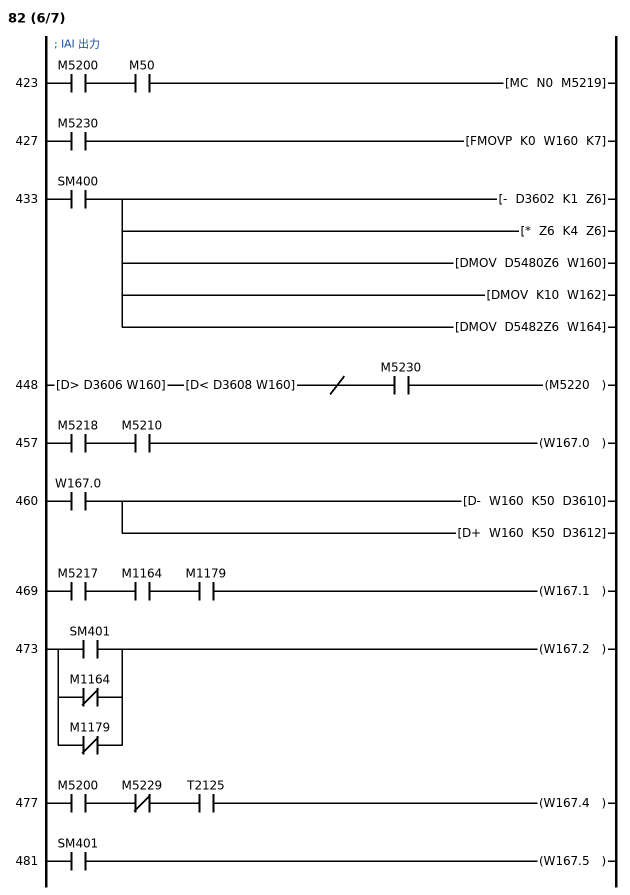
; IAI 出力
423   LD      M5200
      AND     M50
      MC      N0 M5219
427   LD      M5230
      FMOVP   K0 W160 K7
433   LD      SM400
      -       D3602 K1 Z6
      *       Z6 K4 Z6
      DMOV    D5480Z6 W160
      DMOV    K10 W162
      DMOV    D5482Z6 W164
448   LDD>    D3606 W160
      ANDD<   D3608 W160
      INV
      AND     M5230
      OUT     M5220
457   LD      M5218
      AND     M5210
      OUT     W167.0
460   LD      W167.0
      D-      W160 K50 D3610
      D+      W160 K50 D3612
469   LD      M5217
      AND     M1164
      AND     M1179
      OUT     W167.1
473   LD      SM401
      ORI     M1164
      ORI     M1179
      OUT     W167.2
477   LD      M5200
      ANI     M5229
      AND     T2125
      OUT     W167.4
481   LD      SM401
      OUT     W167.5
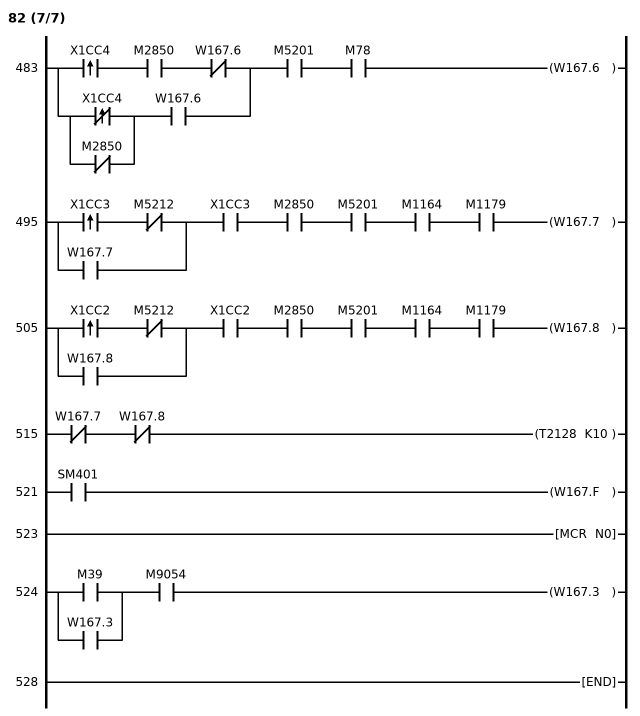
483   LDP     X1CC4
      AND     M2850
      ANI     W167.6
      LDPI    X1CC4
      ORI     M2850
      AND     W167.6
      ORB
      AND     M5201
      AND     M78
      OUT     W167.6
495   LDP     X1CC3
      ANI     M5212
      OR      W167.7
      AND     X1CC3
      AND     M2850
      AND     M5201
      AND     M1164
      AND     M1179
      OUT     W167.7
505   LDP     X1CC2
      ANI     M5212
      OR      W167.8
      AND     X1CC2
      AND     M2850
      AND     M5201
      AND     M1164
      AND     M1179
      OUT     W167.8
515   LDI     W167.7
      ANI     W167.8
      OUT     T2128 K10
521   LD      SM401
      OUT     W167.F
523   MCR     N0
524   LD      M39
      OR      W167.3
      AND     M9054
      OUT     W167.3
528   END
END_PROGRAM

PROGRAM 83
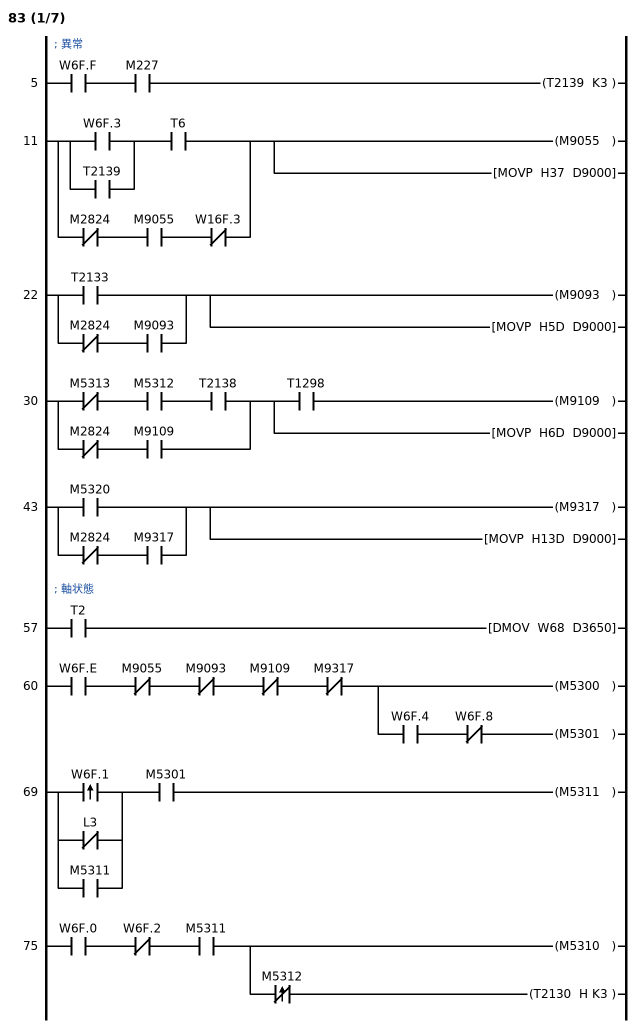
; 異常
5     LD      W6F.F
      AND     M227
      OUT     T2139 K3
11    LD      W6F.3
      OR      T2139
      AND     T6
      LDI     M2824
      AND     M9055
      ANI     W16F.3
      ORB
      OUT     M9055
      MOVP    H37 D9000
22    LD      T2133
      LDI     M2824
      AND     M9093
      ORB
      OUT     M9093
      MOVP    H5D D9000
30    LDI     M5313
      AND     M5312
      AND     T2138
      LDI     M2824
      AND     M9109
      ORB
      MPS
      AND     T1298
      OUT     M9109
      MPP
      MOVP    H6D D9000
43    LD      M5320
      LDI     M2824
      AND     M9317
      ORB
      OUT     M9317
      MOVP    H13D D9000
; 軸状態
57    LD      T2
      DMOV    W68 D3650
60    LD      W6F.E
      ANI     M9055
      ANI     M9093
      ANI     M9109
      ANI     M9317
      OUT     M5300
      AND     W6F.4
      ANI     W6F.8
      OUT     M5301
69    LDP     W6F.1
      ORI     L3
      OR      M5311
      AND     M5301
      OUT     M5311
75    LD      W6F.0
      ANI     W6F.2
      AND     M5311
      OUT     M5310
      ANDPI   M5312
      OUTH    T2130 K3
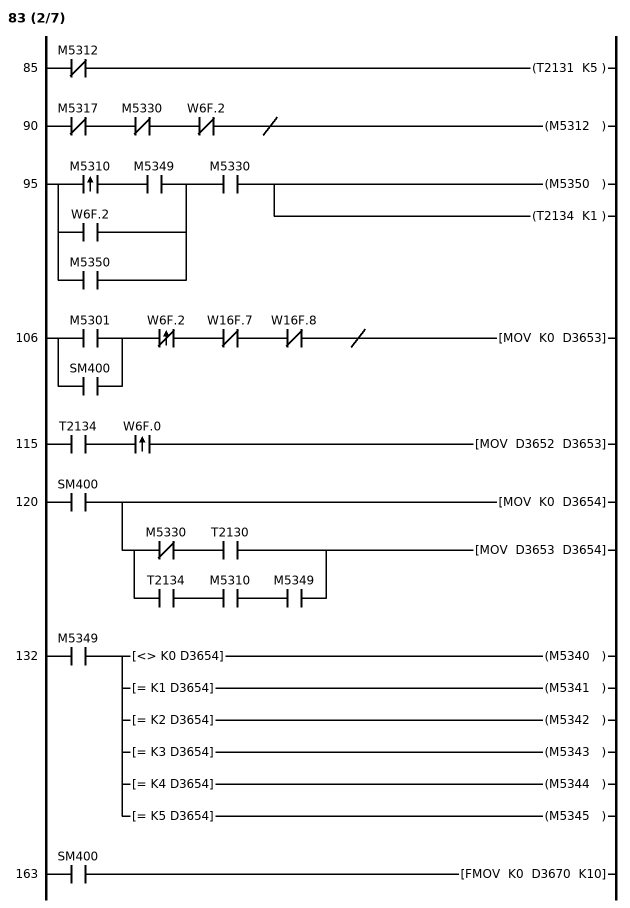
85    LDI     M5312
      OUT     T2131 K5
90    LDI     M5317
      ANI     M5330
      ANI     W6F.2
      INV
      OUT     M5312
95    LDP     M5310
      AND     M5349
      OR      W6F.2
      OR      M5350
      AND     M5330
      OUT     M5350
      OUT     T2134 K1
106   LD      M5301
      OR      SM400
      ANDPI   W6F.2
      ANI     W16F.7
      ANI     W16F.8
      INV
      MOV     K0 D3653
115   LD      T2134
      ANDP    W6F.0
      MOV     D3652 D3653
120   LD      SM400
      MOV     K0 D3654
      LDI     M5330
      AND     T2130
      LD      T2134
      AND     M5310
      AND     M5349
      ORB
      ANB
      MOV     D3653 D3654
132   LD      M5349
      MPS
      AND<>   K0 D3654
      OUT     M5340
      MRD
      AND=    K1 D3654
      OUT     M5341
      MRD
      AND=    K2 D3654
      OUT     M5342
      MRD
      AND=    K3 D3654
      OUT     M5343
      MRD
      AND=    K4 D3654
      OUT     M5344
      MPP
      AND=    K5 D3654
      OUT     M5345
163   LD      SM400
      FMOV    K0 D3670 K10
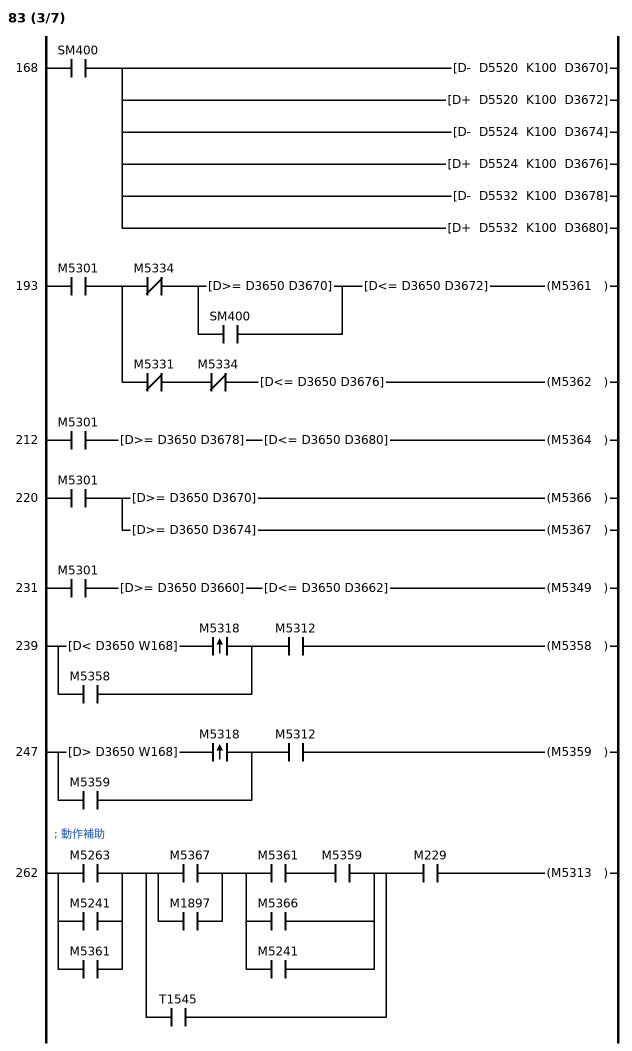
168   LD      SM400
      D-      D5520 K100 D3670
      D+      D5520 K100 D3672
      D-      D5524 K100 D3674
      D+      D5524 K100 D3676
      D-      D5532 K100 D3678
      D+      D5532 K100 D3680
193   LD      M5301
      MPS
      ANI     M5334
      LDD>=   D3650 D3670
      OR      SM400
      ANB
      ANDD<=  D3650 D3672
      OUT     M5361
      MPP
      ANI     M5331
      ANI     M5334
      ANDD<=  D3650 D3676
      OUT     M5362
212   LD      M5301
      ANDD>=  D3650 D3678
      ANDD<=  D3650 D3680
      OUT     M5364
220   LD      M5301
      MPS
      ANDD>=  D3650 D3670
      OUT     M5366
      MPP
      ANDD>=  D3650 D3674
      OUT     M5367
231   LD      M5301
      ANDD>=  D3650 D3660
      ANDD<=  D3650 D3662
      OUT     M5349
239   LDD<    D3650 W168
      ANDP    M5318
      OR      M5358
      AND     M5312
      OUT     M5358
247   LDD>    D3650 W168
      ANDP    M5318
      OR      M5359
      AND     M5312
      OUT     M5359
; 動作補助
262   LD      M5263
      OR      M5241
      OR      M5361
      LD      M5367
      OR      M1897
      LD      M5361
      AND     M5359
      OR      M5366
      OR      M5241
      ANB
      OR      T1545
      ANB
      AND     M229
      OUT     M5313
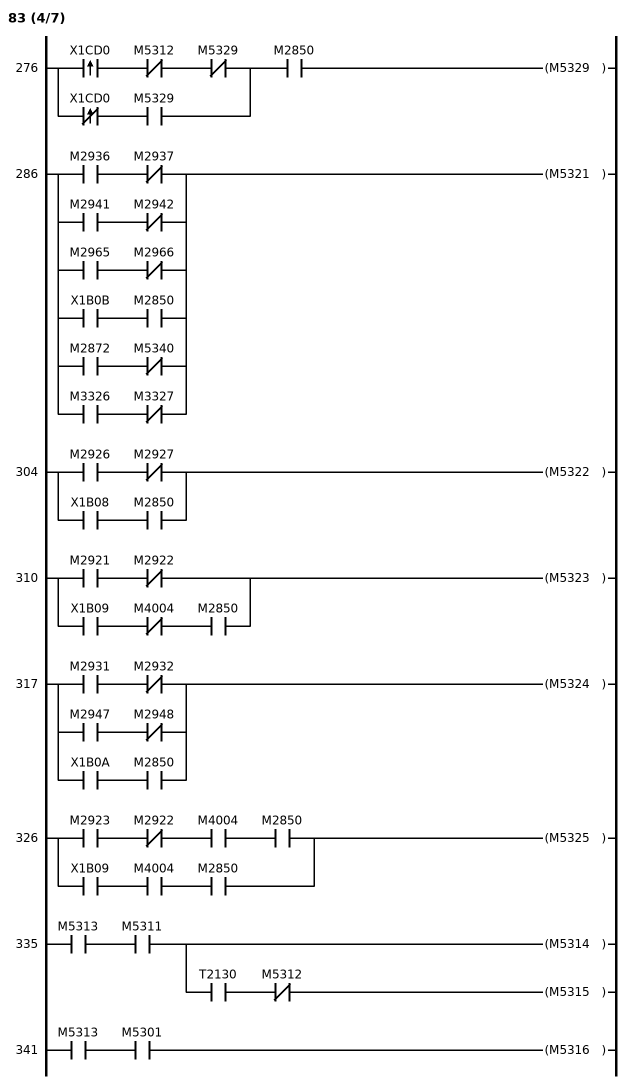
276   LDP     X1CD0
      ANI     M5312
      ANI     M5329
      LDPI    X1CD0
      AND     M5329
      ORB
      AND     M2850
      OUT     M5329
286   LD      M2936
      ANI     M2937
      LD      M2941
      ANI     M2942
      ORB
      LD      M2965
      ANI     M2966
      ORB
      LD      X1B0B
      AND     M2850
      ORB
      LD      M2872
      ANI     M5340
      ORB
      LD      M3326
      ANI     M3327
      ORB
      OUT     M5321
304   LD      M2926
      ANI     M2927
      LD      X1B08
      AND     M2850
      ORB
      OUT     M5322
310   LD      M2921
      ANI     M2922
      LD      X1B09
      ANI     M4004
      AND     M2850
      ORB
      OUT     M5323
317   LD      M2931
      ANI     M2932
      LD      M2947
      ANI     M2948
      ORB
      LD      X1B0A
      AND     M2850
      ORB
      OUT     M5324
326   LD      M2923
      ANI     M2922
      AND     M4004
      AND     M2850
      LD      X1B09
      AND     M4004
      AND     M2850
      ORB
      OUT     M5325
335   LD      M5313
      AND     M5311
      OUT     M5314
      AND     T2130
      ANI     M5312
      OUT     M5315
341   LD      M5313
      AND     M5301
      OUT     M5316
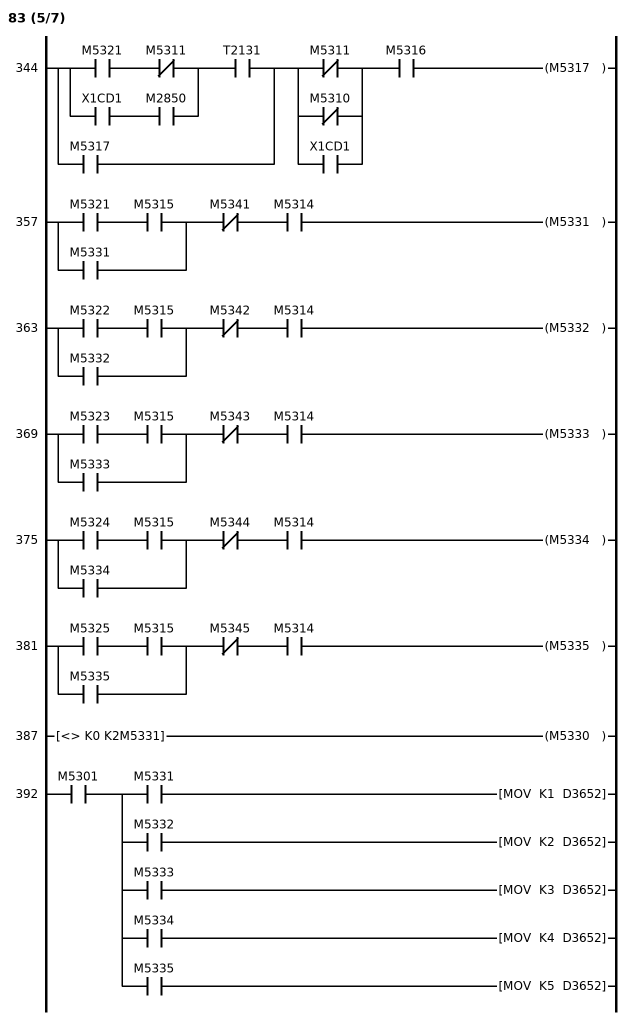
344   LD      M5321
      ANI     M5311
      LD      X1CD1
      AND     M2850
      ORB
      AND     T2131
      OR      M5317
      LDI     M5311
      ORI     M5310
      OR      X1CD1
      ANB
      AND     M5316
      OUT     M5317
357   LD      M5321
      AND     M5315
      OR      M5331
      ANI     M5341
      AND     M5314
      OUT     M5331
363   LD      M5322
      AND     M5315
      OR      M5332
      ANI     M5342
      AND     M5314
      OUT     M5332
369   LD      M5323
      AND     M5315
      OR      M5333
      ANI     M5343
      AND     M5314
      OUT     M5333
375   LD      M5324
      AND     M5315
      OR      M5334
      ANI     M5344
      AND     M5314
      OUT     M5334
381   LD      M5325
      AND     M5315
      OR      M5335
      ANI     M5345
      AND     M5314
      OUT     M5335
387   LD<>    K0 K2M5331
      OUT     M5330
392   LD      M5301
      MPS
      AND     M5331
      MOV     K1 D3652
      MRD
      AND     M5332
      MOV     K2 D3652
      MRD
      AND     M5333
      MOV     K3 D3652
      MRD
      AND     M5334
      MOV     K4 D3652
      MPP
      AND     M5335
      MOV     K5 D3652
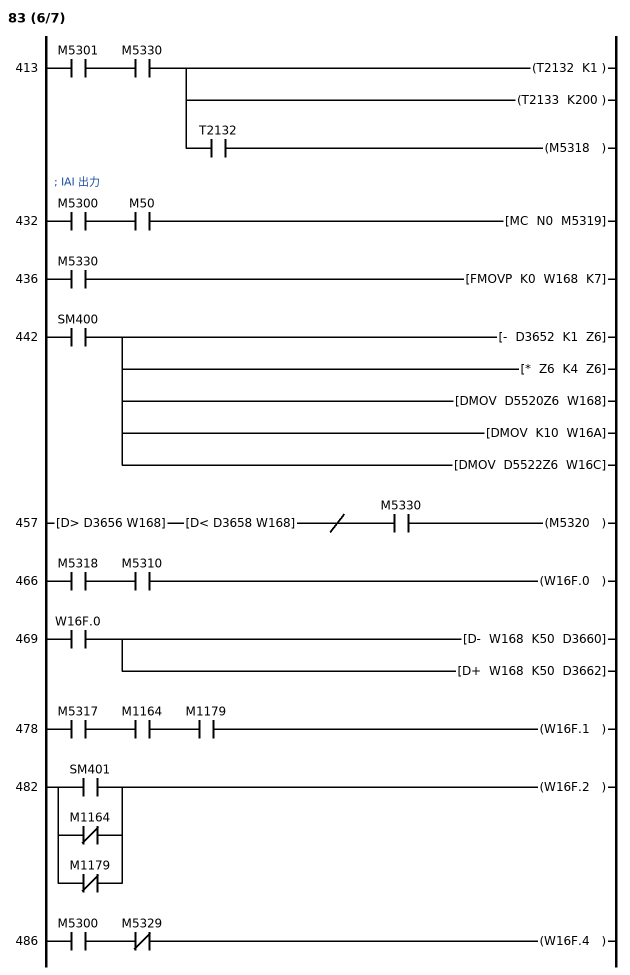
413   LD      M5301
      AND     M5330
      OUT     T2132 K1
      OUT     T2133 K200
      AND     T2132
      OUT     M5318
; IAI 出力
432   LD      M5300
      AND     M50
      MC      N0 M5319
436   LD      M5330
      FMOVP   K0 W168 K7
442   LD      SM400
      -       D3652 K1 Z6
      *       Z6 K4 Z6
      DMOV    D5520Z6 W168
      DMOV    K10 W16A
      DMOV    D5522Z6 W16C
457   LDD>    D3656 W168
      ANDD<   D3658 W168
      INV
      AND     M5330
      OUT     M5320
466   LD      M5318
      AND     M5310
      OUT     W16F.0
469   LD      W16F.0
      D-      W168 K50 D3660
      D+      W168 K50 D3662
478   LD      M5317
      AND     M1164
      AND     M1179
      OUT     W16F.1
482   LD      SM401
      ORI     M1164
      ORI     M1179
      OUT     W16F.2
486   LD      M5300
      ANI     M5329
      OUT     W16F.4
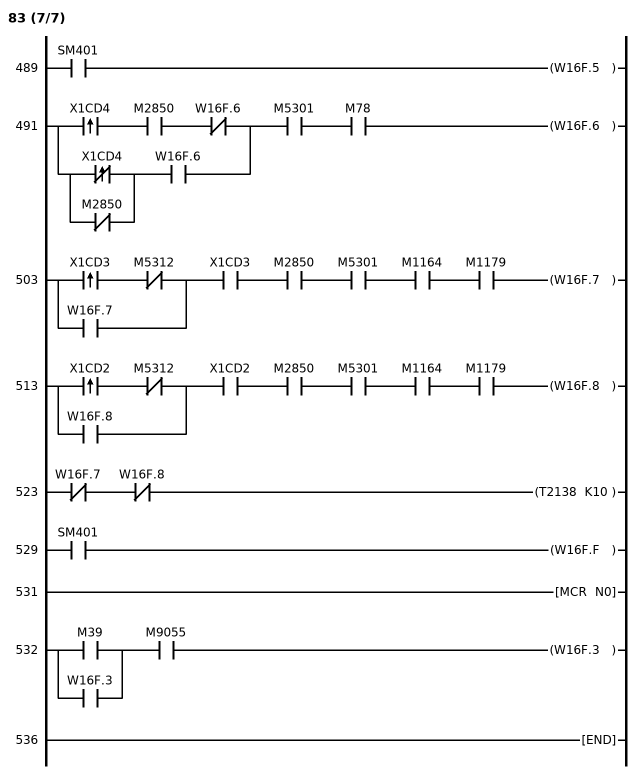
489   LD      SM401
      OUT     W16F.5
491   LDP     X1CD4
      AND     M2850
      ANI     W16F.6
      LDPI    X1CD4
      ORI     M2850
      AND     W16F.6
      ORB
      AND     M5301
      AND     M78
      OUT     W16F.6
503   LDP     X1CD3
      ANI     M5312
      OR      W16F.7
      AND     X1CD3
      AND     M2850
      AND     M5301
      AND     M1164
      AND     M1179
      OUT     W16F.7
513   LDP     X1CD2
      ANI     M5312
      OR      W16F.8
      AND     X1CD2
      AND     M2850
      AND     M5301
      AND     M1164
      AND     M1179
      OUT     W16F.8
523   LDI     W16F.7
      ANI     W16F.8
      OUT     T2138 K10
529   LD      SM401
      OUT     W16F.F
531   MCR     N0
532   LD      M39
      OR      W16F.3
      AND     M9055
      OUT     W16F.3
536   END
END_PROGRAM

PROGRAM 90
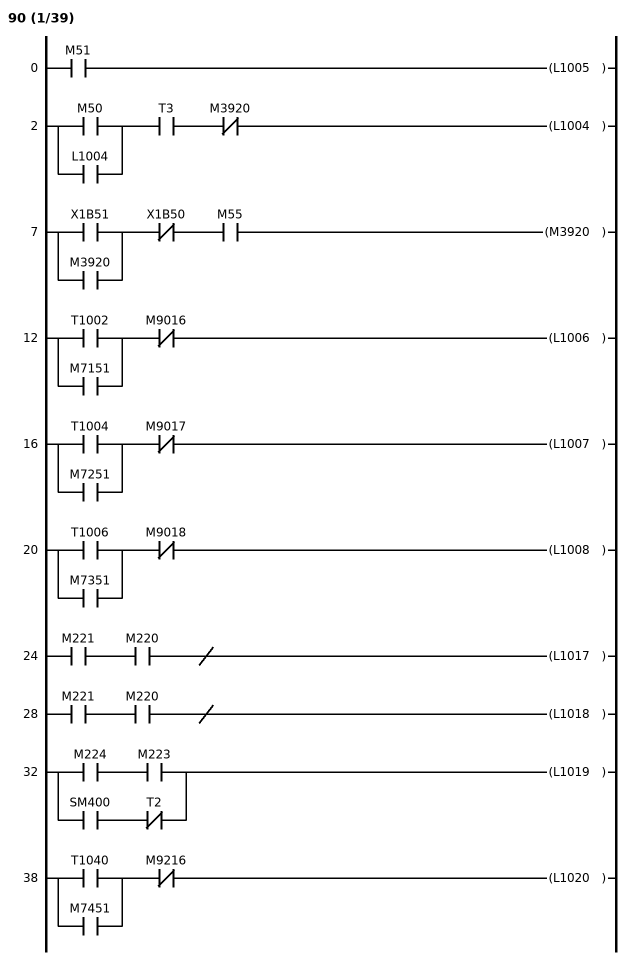
0     LD      M51
      OUT     L1005
2     LD      M50
      OR      L1004
      AND     T3
      ANI     M3920
      OUT     L1004
7     LD      X1B51
      OR      M3920
      ANI     X1B50
      AND     M55
      OUT     M3920
12    LD      T1002
      OR      M7151
      ANI     M9016
      OUT     L1006
16    LD      T1004
      OR      M7251
      ANI     M9017
      OUT     L1007
20    LD      T1006
      OR      M7351
      ANI     M9018
      OUT     L1008
24    LD      M221
      AND     M220
      INV
      OUT     L1017
28    LD      M221
      AND     M220
      INV
      OUT     L1018
32    LD      M224
      AND     M223
      LD      SM400
      ANI     T2
      ORB
      OUT     L1019
38    LD      T1040
      OR      M7451
      ANI     M9216
      OUT     L1020
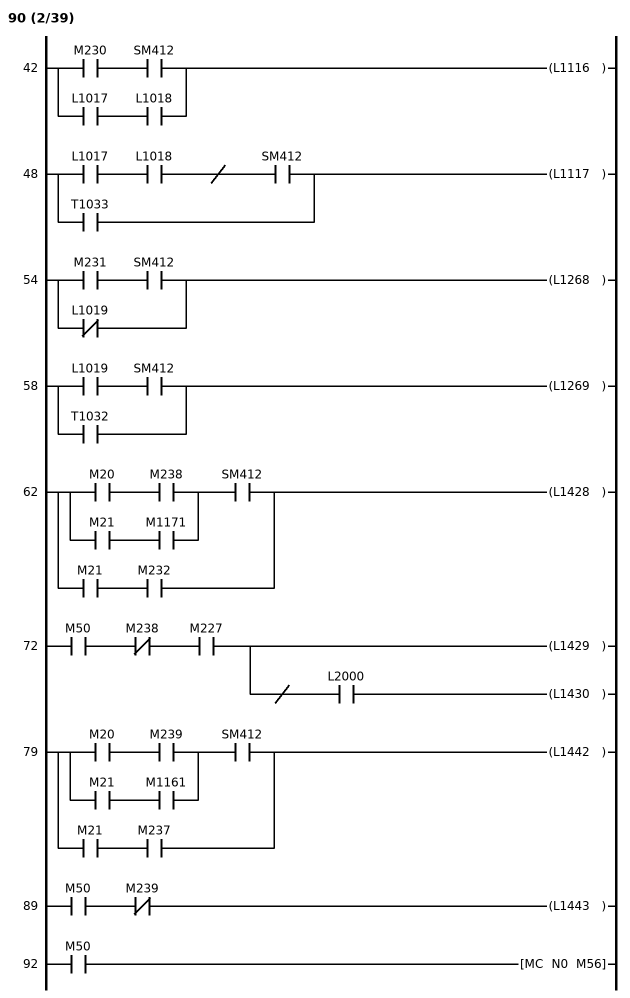
42    LD      M230
      AND     SM412
      LD      L1017
      AND     L1018
      ORB
      OUT     L1116
48    LD      L1017
      AND     L1018
      INV
      AND     SM412
      OR      T1033
      OUT     L1117
54    LD      M231
      AND     SM412
      ORI     L1019
      OUT     L1268
58    LD      L1019
      AND     SM412
      OR      T1032
      OUT     L1269
62    LD      M20
      AND     M238
      LD      M21
      AND     M1171
      ORB
      AND     SM412
      LD      M21
      AND     M232
      ORB
      OUT     L1428
72    LD      M50
      ANI     M238
      AND     M227
      OUT     L1429
      INV
      AND     L2000
      OUT     L1430
79    LD      M20
      AND     M239
      LD      M21
      AND     M1161
      ORB
      AND     SM412
      LD      M21
      AND     M237
      ORB
      OUT     L1442
89    LD      M50
      ANI     M239
      OUT     L1443
92    LD      M50
      MC      N0 M56
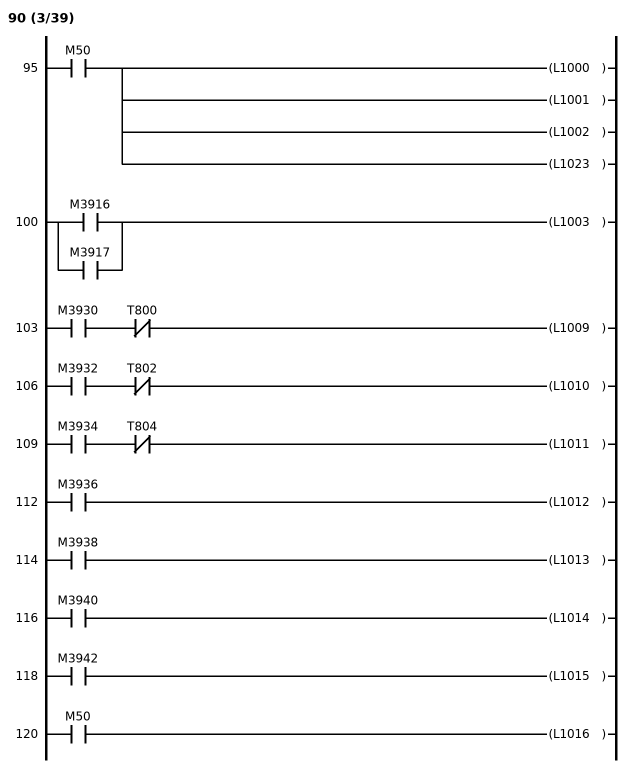
95    LD      M50
      OUT     L1000
      OUT     L1001
      OUT     L1002
      OUT     L1023
100   LD      M3916
      OR      M3917
      OUT     L1003
103   LD      M3930
      ANI     T800
      OUT     L1009
106   LD      M3932
      ANI     T802
      OUT     L1010
109   LD      M3934
      ANI     T804
      OUT     L1011
112   LD      M3936
      OUT     L1012
114   LD      M3938
      OUT     L1013
116   LD      M3940
      OUT     L1014
118   LD      M3942
      OUT     L1015
120   LD      M50
      OUT     L1016
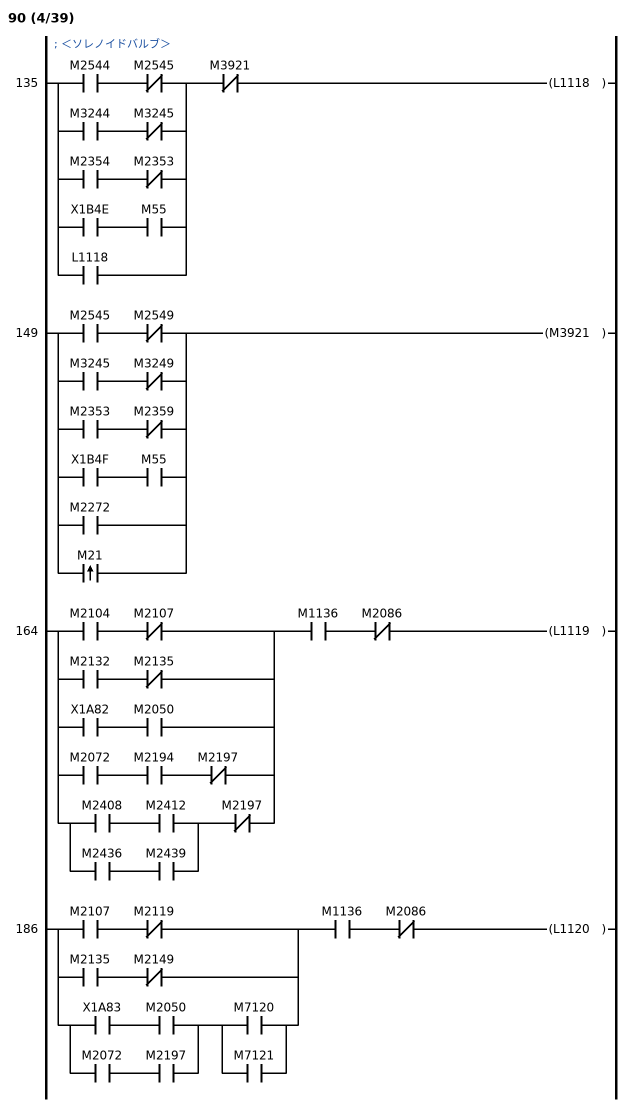
; ＜ソレノイドバルブ＞
135   LD      M2544
      ANI     M2545
      LD      M3244
      ANI     M3245
      ORB
      LD      M2354
      ANI     M2353
      ORB
      LD      X1B4E
      AND     M55
      ORB
      OR      L1118
      ANI     M3921
      OUT     L1118
149   LD      M2545
      ANI     M2549
      LD      M3245
      ANI     M3249
      ORB
      LD      M2353
      ANI     M2359
      ORB
      LD      X1B4F
      AND     M55
      ORB
      OR      M2272
      ORP     M21
      OUT     M3921
164   LD      M2104
      ANI     M2107
      LD      M2132
      ANI     M2135
      ORB
      LD      X1A82
      AND     M2050
      ORB
      LD      M2072
      AND     M2194
      ANI     M2197
      ORB
      LD      M2408
      AND     M2412
      LD      M2436
      AND     M2439
      ORB
      ANI     M2197
      ORB
      AND     M1136
      ANI     M2086
      OUT     L1119
186   LD      M2107
      ANI     M2119
      LD      M2135
      ANI     M2149
      ORB
      LD      X1A83
      AND     M2050
      LD      M2072
      AND     M2197
      ORB
      LD      M7120
      OR      M7121
      ANB
      ORB
      AND     M1136
      ANI     M2086
      OUT     L1120
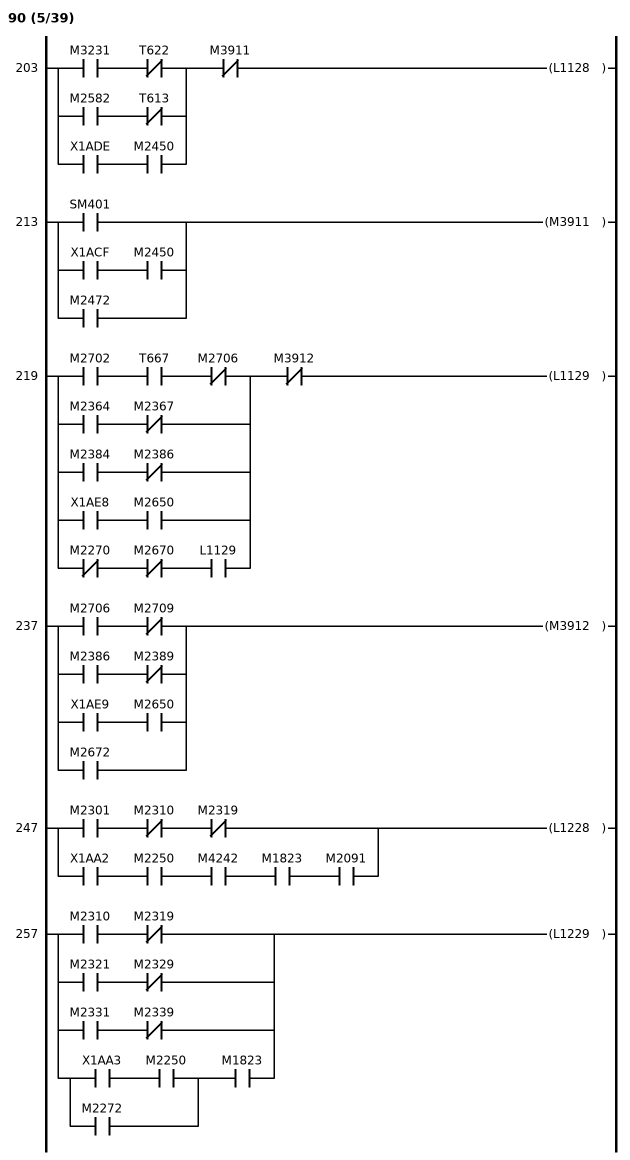
203   LD      M3231
      ANI     T622
      LD      M2582
      ANI     T613
      ORB
      LD      X1ADE
      AND     M2450
      ORB
      ANI     M3911
      OUT     L1128
213   LD      SM401
      LD      X1ACF
      AND     M2450
      ORB
      OR      M2472
      OUT     M3911
219   LD      M2702
      AND     T667
      ANI     M2706
      LD      M2364
      ANI     M2367
      ORB
      LD      M2384
      ANI     M2386
      ORB
      LD      X1AE8
      AND     M2650
      ORB
      LDI     M2270
      ANI     M2670
      AND     L1129
      ORB
      ANI     M3912
      OUT     L1129
237   LD      M2706
      ANI     M2709
      LD      M2386
      ANI     M2389
      ORB
      LD      X1AE9
      AND     M2650
      ORB
      OR      M2672
      OUT     M3912
247   LD      M2301
      ANI     M2310
      ANI     M2319
      LD      X1AA2
      AND     M2250
      AND     M4242
      AND     M1823
      AND     M2091
      ORB
      OUT     L1228
257   LD      M2310
      ANI     M2319
      LD      M2321
      ANI     M2329
      ORB
      LD      M2331
      ANI     M2339
      ORB
      LD      X1AA3
      AND     M2250
      OR      M2272
      AND     M1823
      ORB
      OUT     L1229
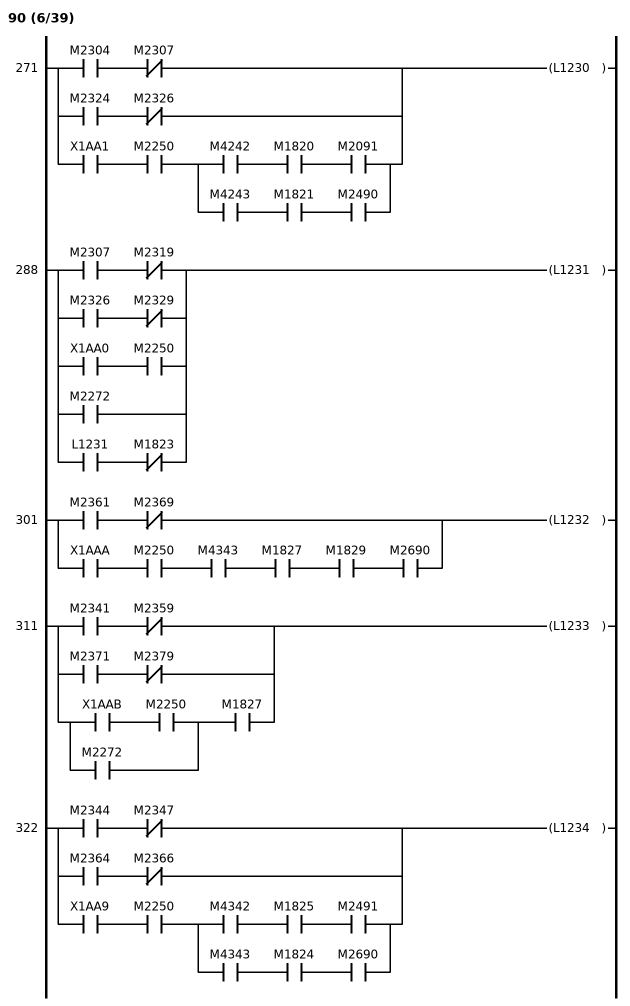
271   LD      M2304
      ANI     M2307
      LD      M2324
      ANI     M2326
      ORB
      LD      X1AA1
      AND     M2250
      LD      M4242
      AND     M1820
      AND     M2091
      LD      M4243
      AND     M1821
      AND     M2490
      ORB
      ANB
      ORB
      OUT     L1230
288   LD      M2307
      ANI     M2319
      LD      M2326
      ANI     M2329
      ORB
      LD      X1AA0
      AND     M2250
      ORB
      OR      M2272
      LD      L1231
      ANI     M1823
      ORB
      OUT     L1231
301   LD      M2361
      ANI     M2369
      LD      X1AAA
      AND     M2250
      AND     M4343
      AND     M1827
      AND     M1829
      AND     M2690
      ORB
      OUT     L1232
311   LD      M2341
      ANI     M2359
      LD      M2371
      ANI     M2379
      ORB
      LD      X1AAB
      AND     M2250
      OR      M2272
      AND     M1827
      ORB
      OUT     L1233
322   LD      M2344
      ANI     M2347
      LD      M2364
      ANI     M2366
      ORB
      LD      X1AA9
      AND     M2250
      LD      M4342
      AND     M1825
      AND     M2491
      LD      M4343
      AND     M1824
      AND     M2690
      ORB
      ANB
      ORB
      OUT     L1234
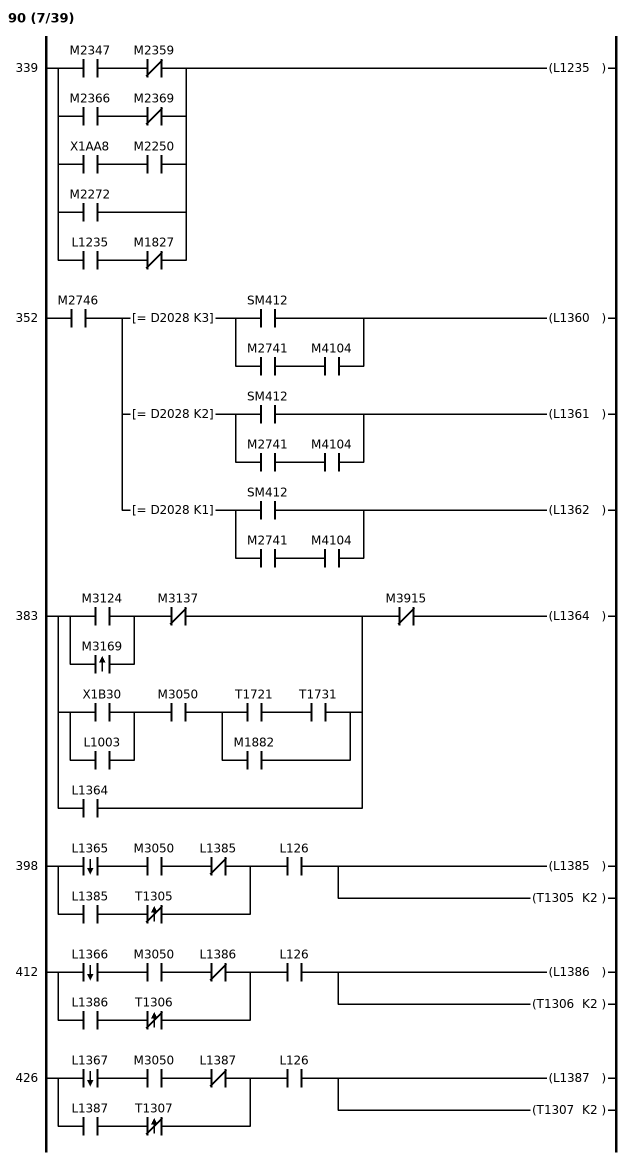
339   LD      M2347
      ANI     M2359
      LD      M2366
      ANI     M2369
      ORB
      LD      X1AA8
      AND     M2250
      ORB
      OR      M2272
      LD      L1235
      ANI     M1827
      ORB
      OUT     L1235
352   LD      M2746
      MPS
      AND=    D2028 K3
      LD      SM412
      LD      M2741
      AND     M4104
      ORB
      ANB
      OUT     L1360
      MRD
      AND=    D2028 K2
      LD      SM412
      LD      M2741
      AND     M4104
      ORB
      ANB
      OUT     L1361
      MPP
      AND=    D2028 K1
      LD      SM412
      LD      M2741
      AND     M4104
      ORB
      ANB
      OUT     L1362
383   LD      M3124
      ORP     M3169
      ANI     M3137
      LD      X1B30
      OR      L1003
      AND     M3050
      LD      T1721
      AND     T1731
      OR      M1882
      ANB
      ORB
      OR      L1364
      ANI     M3915
      OUT     L1364
398   LDF     L1365
      AND     M3050
      ANI     L1385
      LD      L1385
      ANDPI   T1305
      ORB
      AND     L126
      OUT     L1385
      OUT     T1305 K2
412   LDF     L1366
      AND     M3050
      ANI     L1386
      LD      L1386
      ANDPI   T1306
      ORB
      AND     L126
      OUT     L1386
      OUT     T1306 K2
426   LDF     L1367
      AND     M3050
      ANI     L1387
      LD      L1387
      ANDPI   T1307
      ORB
      AND     L126
      OUT     L1387
      OUT     T1307 K2
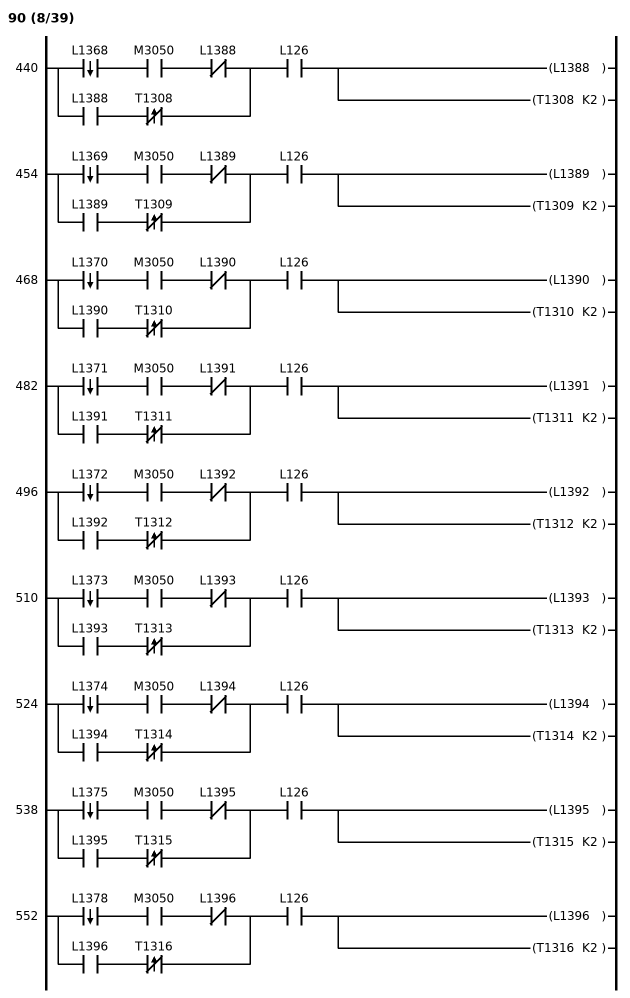
440   LDF     L1368
      AND     M3050
      ANI     L1388
      LD      L1388
      ANDPI   T1308
      ORB
      AND     L126
      OUT     L1388
      OUT     T1308 K2
454   LDF     L1369
      AND     M3050
      ANI     L1389
      LD      L1389
      ANDPI   T1309
      ORB
      AND     L126
      OUT     L1389
      OUT     T1309 K2
468   LDF     L1370
      AND     M3050
      ANI     L1390
      LD      L1390
      ANDPI   T1310
      ORB
      AND     L126
      OUT     L1390
      OUT     T1310 K2
482   LDF     L1371
      AND     M3050
      ANI     L1391
      LD      L1391
      ANDPI   T1311
      ORB
      AND     L126
      OUT     L1391
      OUT     T1311 K2
496   LDF     L1372
      AND     M3050
      ANI     L1392
      LD      L1392
      ANDPI   T1312
      ORB
      AND     L126
      OUT     L1392
      OUT     T1312 K2
510   LDF     L1373
      AND     M3050
      ANI     L1393
      LD      L1393
      ANDPI   T1313
      ORB
      AND     L126
      OUT     L1393
      OUT     T1313 K2
524   LDF     L1374
      AND     M3050
      ANI     L1394
      LD      L1394
      ANDPI   T1314
      ORB
      AND     L126
      OUT     L1394
      OUT     T1314 K2
538   LDF     L1375
      AND     M3050
      ANI     L1395
      LD      L1395
      ANDPI   T1315
      ORB
      AND     L126
      OUT     L1395
      OUT     T1315 K2
552   LDF     L1378
      AND     M3050
      ANI     L1396
      LD      L1396
      ANDPI   T1316
      ORB
      AND     L126
      OUT     L1396
      OUT     T1316 K2
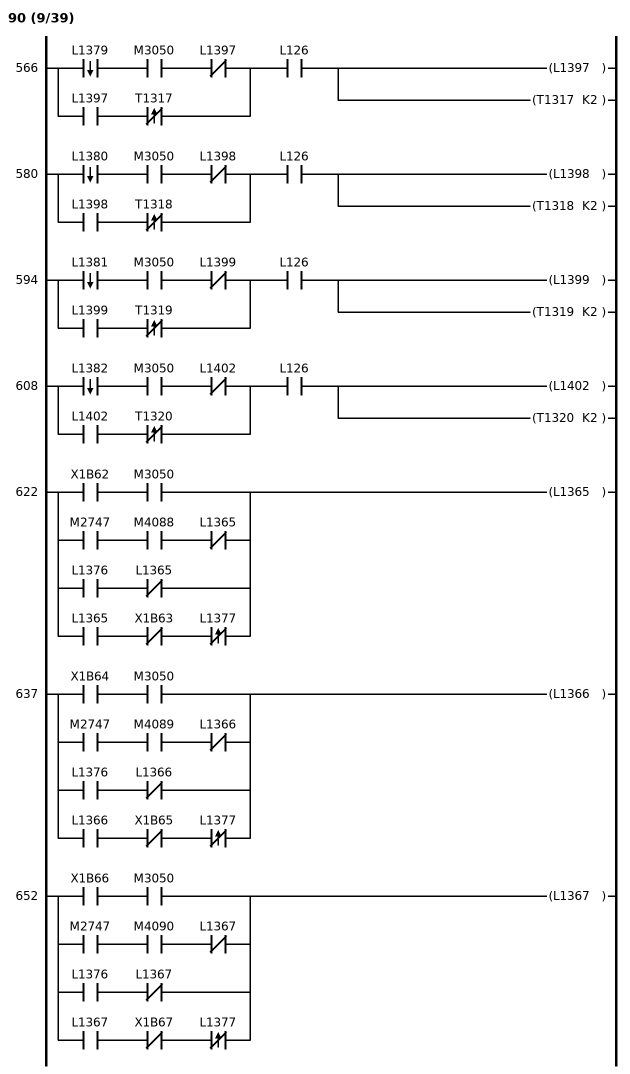
566   LDF     L1379
      AND     M3050
      ANI     L1397
      LD      L1397
      ANDPI   T1317
      ORB
      AND     L126
      OUT     L1397
      OUT     T1317 K2
580   LDF     L1380
      AND     M3050
      ANI     L1398
      LD      L1398
      ANDPI   T1318
      ORB
      AND     L126
      OUT     L1398
      OUT     T1318 K2
594   LDF     L1381
      AND     M3050
      ANI     L1399
      LD      L1399
      ANDPI   T1319
      ORB
      AND     L126
      OUT     L1399
      OUT     T1319 K2
608   LDF     L1382
      AND     M3050
      ANI     L1402
      LD      L1402
      ANDPI   T1320
      ORB
      AND     L126
      OUT     L1402
      OUT     T1320 K2
622   LD      X1B62
      AND     M3050
      LD      M2747
      AND     M4088
      ANI     L1365
      ORB
      LD      L1376
      ANI     L1365
      ORB
      LD      L1365
      ANI     X1B63
      ANDPI   L1377
      ORB
      OUT     L1365
637   LD      X1B64
      AND     M3050
      LD      M2747
      AND     M4089
      ANI     L1366
      ORB
      LD      L1376
      ANI     L1366
      ORB
      LD      L1366
      ANI     X1B65
      ANDPI   L1377
      ORB
      OUT     L1366
652   LD      X1B66
      AND     M3050
      LD      M2747
      AND     M4090
      ANI     L1367
      ORB
      LD      L1376
      ANI     L1367
      ORB
      LD      L1367
      ANI     X1B67
      ANDPI   L1377
      ORB
      OUT     L1367
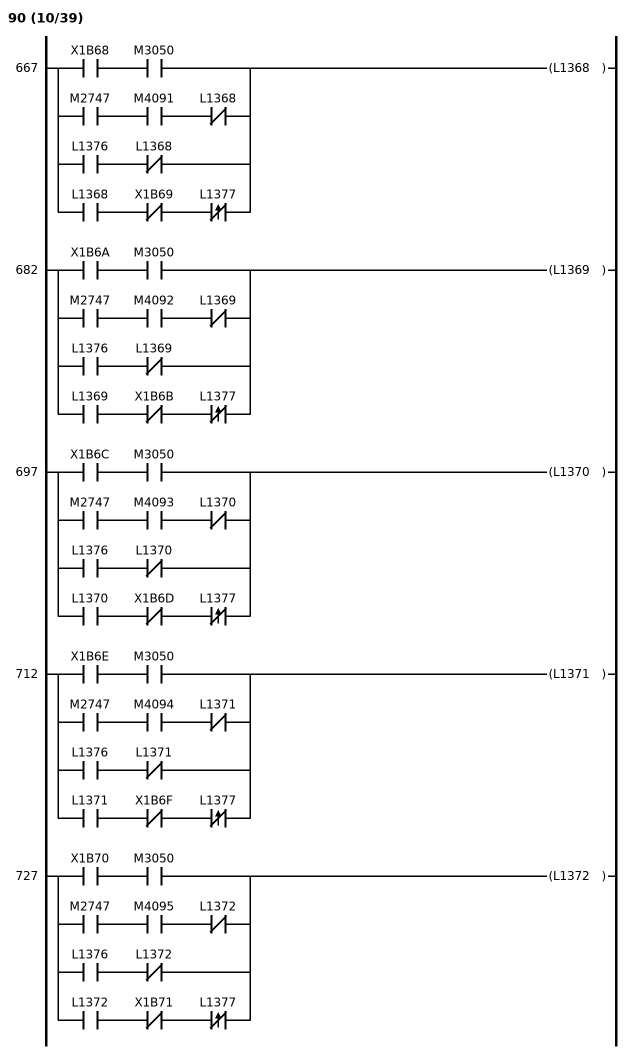
667   LD      X1B68
      AND     M3050
      LD      M2747
      AND     M4091
      ANI     L1368
      ORB
      LD      L1376
      ANI     L1368
      ORB
      LD      L1368
      ANI     X1B69
      ANDPI   L1377
      ORB
      OUT     L1368
682   LD      X1B6A
      AND     M3050
      LD      M2747
      AND     M4092
      ANI     L1369
      ORB
      LD      L1376
      ANI     L1369
      ORB
      LD      L1369
      ANI     X1B6B
      ANDPI   L1377
      ORB
      OUT     L1369
697   LD      X1B6C
      AND     M3050
      LD      M2747
      AND     M4093
      ANI     L1370
      ORB
      LD      L1376
      ANI     L1370
      ORB
      LD      L1370
      ANI     X1B6D
      ANDPI   L1377
      ORB
      OUT     L1370
712   LD      X1B6E
      AND     M3050
      LD      M2747
      AND     M4094
      ANI     L1371
      ORB
      LD      L1376
      ANI     L1371
      ORB
      LD      L1371
      ANI     X1B6F
      ANDPI   L1377
      ORB
      OUT     L1371
727   LD      X1B70
      AND     M3050
      LD      M2747
      AND     M4095
      ANI     L1372
      ORB
      LD      L1376
      ANI     L1372
      ORB
      LD      L1372
      ANI     X1B71
      ANDPI   L1377
      ORB
      OUT     L1372
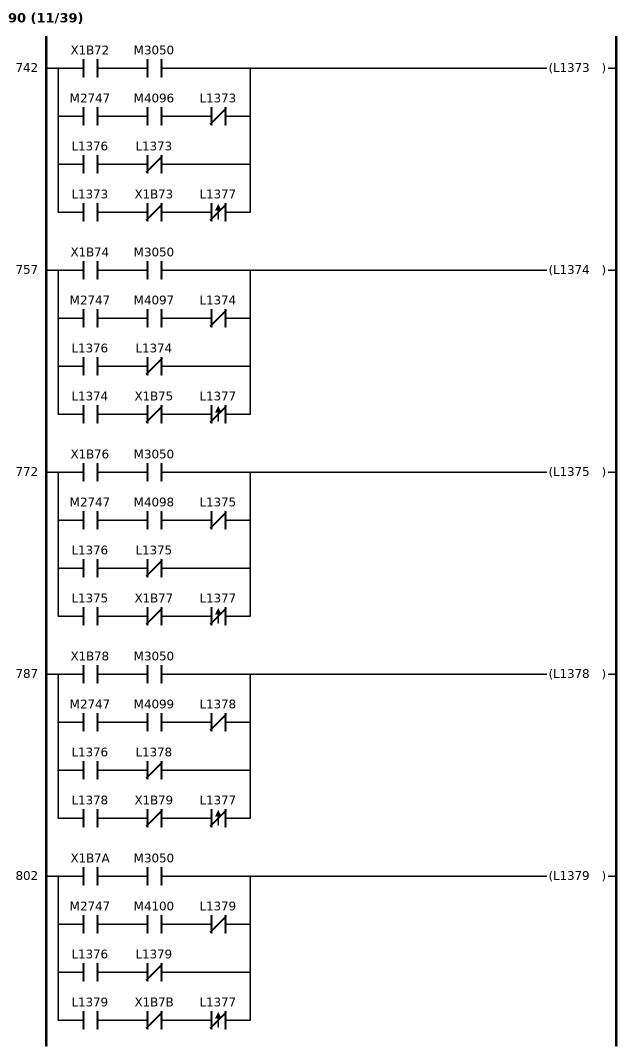
742   LD      X1B72
      AND     M3050
      LD      M2747
      AND     M4096
      ANI     L1373
      ORB
      LD      L1376
      ANI     L1373
      ORB
      LD      L1373
      ANI     X1B73
      ANDPI   L1377
      ORB
      OUT     L1373
757   LD      X1B74
      AND     M3050
      LD      M2747
      AND     M4097
      ANI     L1374
      ORB
      LD      L1376
      ANI     L1374
      ORB
      LD      L1374
      ANI     X1B75
      ANDPI   L1377
      ORB
      OUT     L1374
772   LD      X1B76
      AND     M3050
      LD      M2747
      AND     M4098
      ANI     L1375
      ORB
      LD      L1376
      ANI     L1375
      ORB
      LD      L1375
      ANI     X1B77
      ANDPI   L1377
      ORB
      OUT     L1375
787   LD      X1B78
      AND     M3050
      LD      M2747
      AND     M4099
      ANI     L1378
      ORB
      LD      L1376
      ANI     L1378
      ORB
      LD      L1378
      ANI     X1B79
      ANDPI   L1377
      ORB
      OUT     L1378
802   LD      X1B7A
      AND     M3050
      LD      M2747
      AND     M4100
      ANI     L1379
      ORB
      LD      L1376
      ANI     L1379
      ORB
      LD      L1379
      ANI     X1B7B
      ANDPI   L1377
      ORB
      OUT     L1379
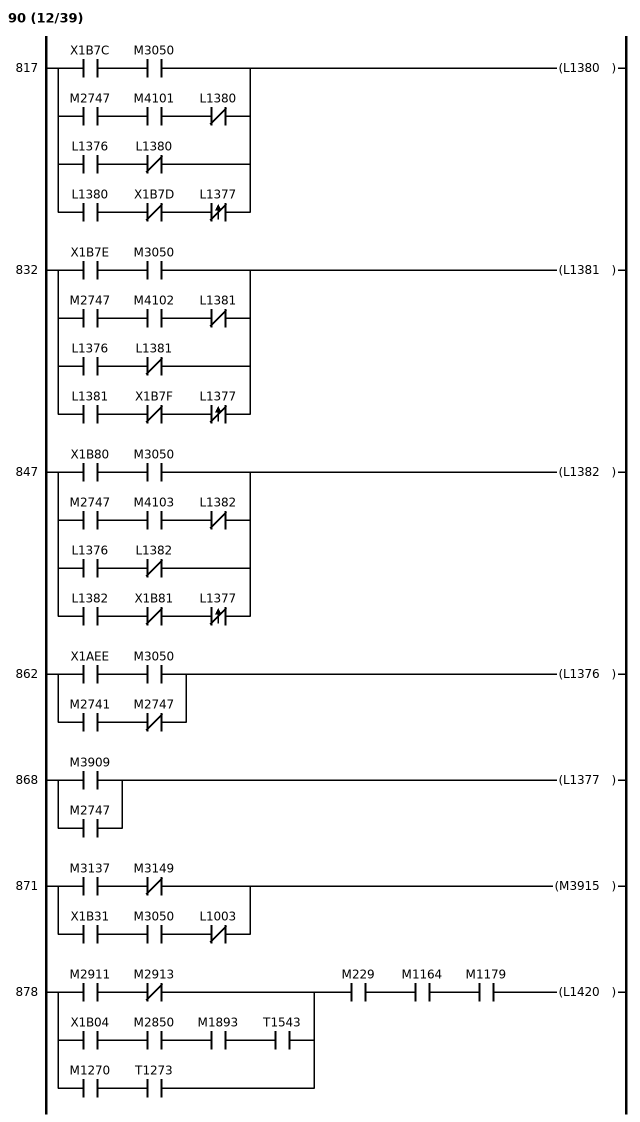
817   LD      X1B7C
      AND     M3050
      LD      M2747
      AND     M4101
      ANI     L1380
      ORB
      LD      L1376
      ANI     L1380
      ORB
      LD      L1380
      ANI     X1B7D
      ANDPI   L1377
      ORB
      OUT     L1380
832   LD      X1B7E
      AND     M3050
      LD      M2747
      AND     M4102
      ANI     L1381
      ORB
      LD      L1376
      ANI     L1381
      ORB
      LD      L1381
      ANI     X1B7F
      ANDPI   L1377
      ORB
      OUT     L1381
847   LD      X1B80
      AND     M3050
      LD      M2747
      AND     M4103
      ANI     L1382
      ORB
      LD      L1376
      ANI     L1382
      ORB
      LD      L1382
      ANI     X1B81
      ANDPI   L1377
      ORB
      OUT     L1382
862   LD      X1AEE
      AND     M3050
      LD      M2741
      ANI     M2747
      ORB
      OUT     L1376
868   LD      M3909
      OR      M2747
      OUT     L1377
871   LD      M3137
      ANI     M3149
      LD      X1B31
      AND     M3050
      ANI     L1003
      ORB
      OUT     M3915
878   LD      M2911
      ANI     M2913
      LD      X1B04
      AND     M2850
      AND     M1893
      AND     T1543
      ORB
      LD      M1270
      AND     T1273
      ORB
      AND     M229
      AND     M1164
      AND     M1179
      OUT     L1420
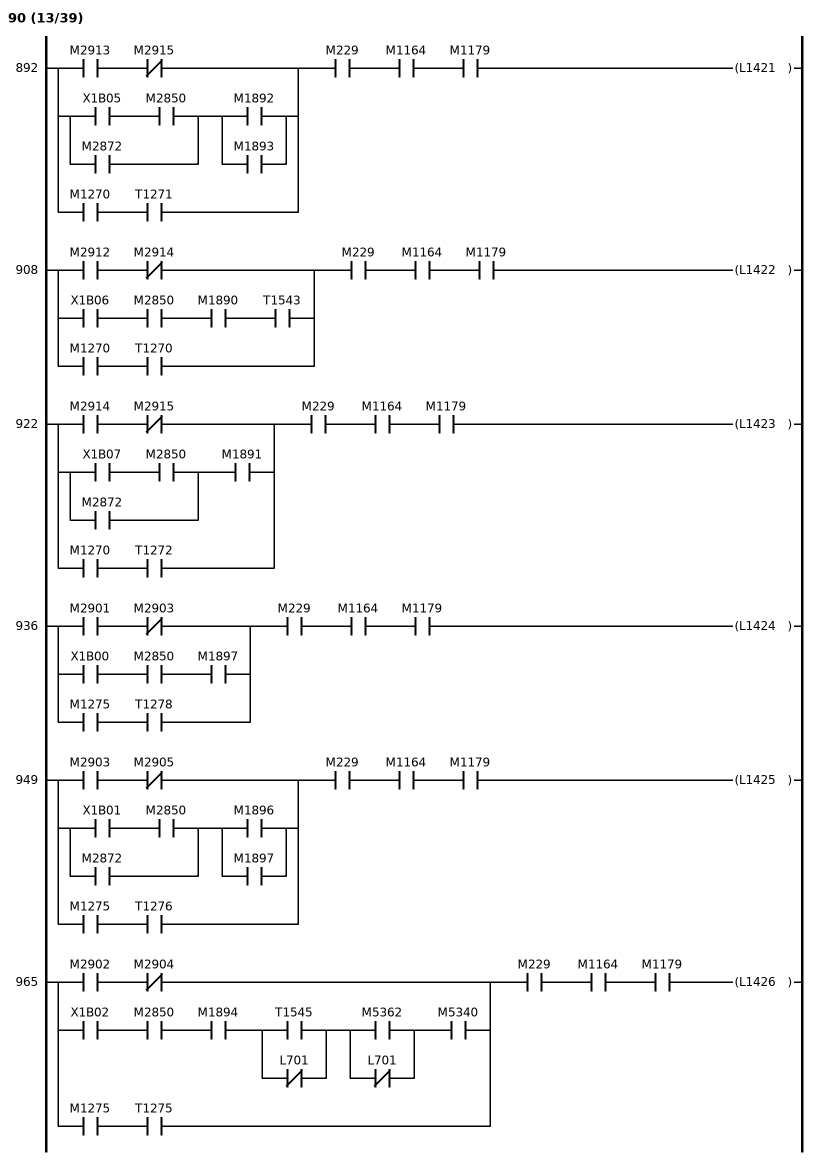
892   LD      M2913
      ANI     M2915
      LD      X1B05
      AND     M2850
      OR      M2872
      LD      M1892
      OR      M1893
      ANB
      ORB
      LD      M1270
      AND     T1271
      ORB
      AND     M229
      AND     M1164
      AND     M1179
      OUT     L1421
908   LD      M2912
      ANI     M2914
      LD      X1B06
      AND     M2850
      AND     M1890
      AND     T1543
      ORB
      LD      M1270
      AND     T1270
      ORB
      AND     M229
      AND     M1164
      AND     M1179
      OUT     L1422
922   LD      M2914
      ANI     M2915
      LD      X1B07
      AND     M2850
      OR      M2872
      AND     M1891
      ORB
      LD      M1270
      AND     T1272
      ORB
      AND     M229
      AND     M1164
      AND     M1179
      OUT     L1423
936   LD      M2901
      ANI     M2903
      LD      X1B00
      AND     M2850
      AND     M1897
      ORB
      LD      M1275
      AND     T1278
      ORB
      AND     M229
      AND     M1164
      AND     M1179
      OUT     L1424
949   LD      M2903
      ANI     M2905
      LD      X1B01
      AND     M2850
      OR      M2872
      LD      M1896
      OR      M1897
      ANB
      ORB
      LD      M1275
      AND     T1276
      ORB
      AND     M229
      AND     M1164
      AND     M1179
      OUT     L1425
965   LD      M2902
      ANI     M2904
      LD      X1B02
      AND     M2850
      AND     M1894
      LD      T1545
      ORI     L701
      ANB
      LD      M5362
      ORI     L701
      ANB
      AND     M5340
      ORB
      LD      M1275
      AND     T1275
      ORB
      AND     M229
      AND     M1164
      AND     M1179
      OUT     L1426
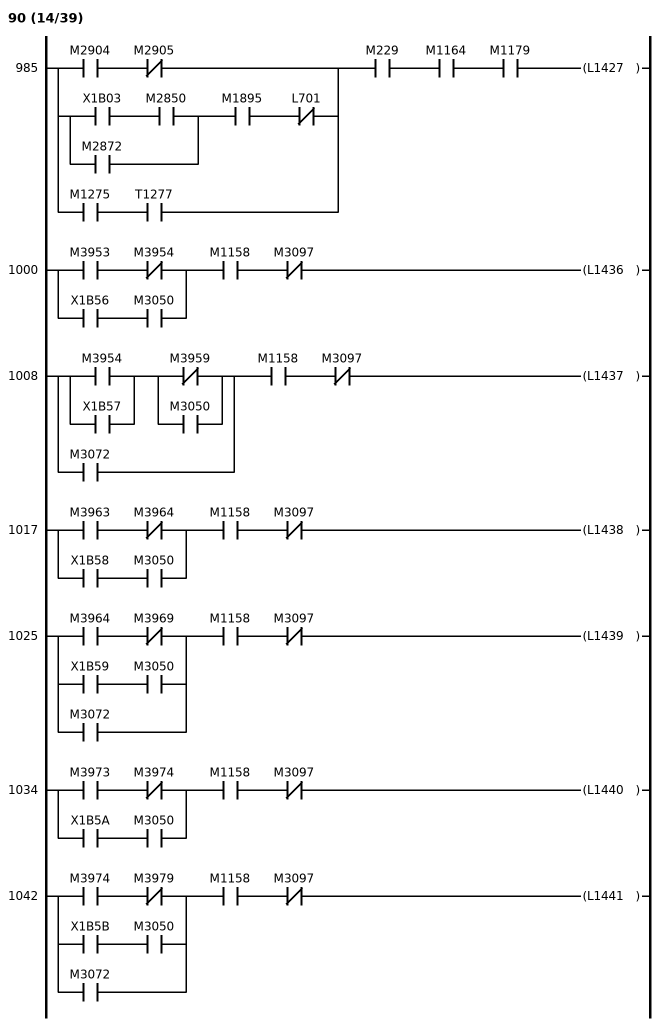
985   LD      M2904
      ANI     M2905
      LD      X1B03
      AND     M2850
      OR      M2872
      AND     M1895
      ANI     L701
      ORB
      LD      M1275
      AND     T1277
      ORB
      AND     M229
      AND     M1164
      AND     M1179
      OUT     L1427
1000  LD      M3953
      ANI     M3954
      LD      X1B56
      AND     M3050
      ORB
      AND     M1158
      ANI     M3097
      OUT     L1436
1008  LD      M3954
      OR      X1B57
      LDI     M3959
      OR      M3050
      ANB
      OR      M3072
      AND     M1158
      ANI     M3097
      OUT     L1437
1017  LD      M3963
      ANI     M3964
      LD      X1B58
      AND     M3050
      ORB
      AND     M1158
      ANI     M3097
      OUT     L1438
1025  LD      M3964
      ANI     M3969
      LD      X1B59
      AND     M3050
      ORB
      OR      M3072
      AND     M1158
      ANI     M3097
      OUT     L1439
1034  LD      M3973
      ANI     M3974
      LD      X1B5A
      AND     M3050
      ORB
      AND     M1158
      ANI     M3097
      OUT     L1440
1042  LD      M3974
      ANI     M3979
      LD      X1B5B
      AND     M3050
      ORB
      OR      M3072
      AND     M1158
      ANI     M3097
      OUT     L1441
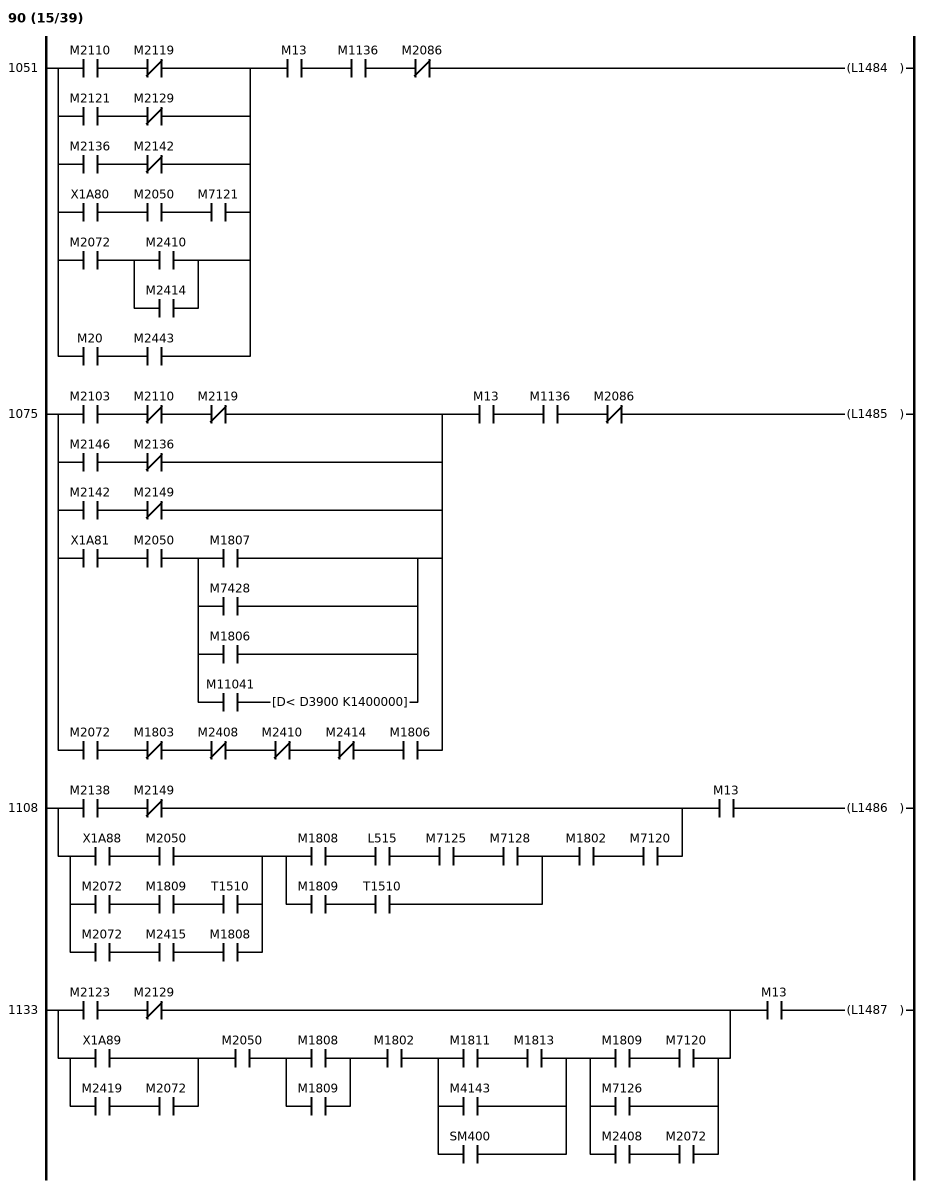
1051  LD      M2110
      ANI     M2119
      LD      M2121
      ANI     M2129
      ORB
      LD      M2136
      ANI     M2142
      ORB
      LD      X1A80
      AND     M2050
      AND     M7121
      ORB
      LD      M2072
      LD      M2410
      OR      M2414
      ANB
      ORB
      LD      M20
      AND     M2443
      ORB
      AND     M13
      AND     M1136
      ANI     M2086
      OUT     L1484
1075  LD      M2103
      ANI     M2110
      ANI     M2119
      LD      M2146
      ANI     M2136
      ORB
      LD      M2142
      ANI     M2149
      ORB
      LD      X1A81
      AND     M2050
      LD      M1807
      OR      M7428
      OR      M1806
      LD      M11041
      ANDD<   D3900 K1400000
      ORB
      ANB
      ORB
      LD      M2072
      ANI     M1803
      ANI     M2408
      ANI     M2410
      ANI     M2414
      AND     M1806
      ORB
      AND     M13
      AND     M1136
      ANI     M2086
      OUT     L1485
1108  LD      M2138
      ANI     M2149
      LD      X1A88
      AND     M2050
      LD      M2072
      AND     M1809
      AND     T1510
      ORB
      LD      M2072
      AND     M2415
      AND     M1808
      ORB
      LD      M1808
      AND     L515
      AND     M7125
      AND     M7128
      LD      M1809
      AND     T1510
      ORB
      ANB
      AND     M1802
      AND     M7120
      ORB
      AND     M13
      OUT     L1486
1133  LD      M2123
      ANI     M2129
      LD      X1A89
      LD      M2419
      AND     M2072
      ORB
      AND     M2050
      LD      M1808
      OR      M1809
      ANB
      AND     M1802
      LD      M1811
      AND     M1813
      OR      M4143
      OR      SM400
      ANB
      LD      M1809
      AND     M7120
      OR      M7126
      LD      M2408
      AND     M2072
      ORB
      ANB
      ORB
      AND     M13
      OUT     L1487
